FUNCTION_BLOCK Master_TEST (* Composite Function Block Type *)
  (* Standard: 61499-2 *)
  (* Version 0.2, 2003-12-05, JHC, Rockwell Automation, Renamed from NEWCOMPFB. *)
  (* Version 0.1, 2002-01-08, JHC, Rockwell Automation, Added DLY FB as example. *)
  (* Version 0.0, 2000-05-27, JHC, Rockwell Automation *)
  (* Compiler header: package fb.rt.pnp; *)
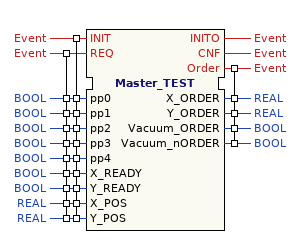
  EVENT_INPUT
    INIT WITH pp0, pp1, pp2, pp3, pp4, X_READY, Y_READY, X_POS, Y_POS; (* Initialization Request *)
    REQ WITH pp0, pp1, pp2, pp3, pp4, X_READY, Y_READY, X_POS, Y_POS; (* Normal Execution Request *)
  END_EVENT
  EVENT_OUTPUT
    INITO; (* Initialization Confirm *)
    CNF; (* Execution Confirmation *)
    Order WITH X_ORDER, Y_ORDER, Vacuum_ORDER, Vacuum_nORDER;
  END_EVENT
  VAR_INPUT
    pp0 : BOOL;
    pp1 : BOOL;
    pp2 : BOOL;
    pp3 : BOOL;
    pp4 : BOOL;
    X_READY : BOOL;
    Y_READY : BOOL;
    X_POS : REAL;
    Y_POS : REAL;
  END_VAR
  VAR_OUTPUT
    X_ORDER : REAL;
    Y_ORDER : REAL;
    Vacuum_ORDER : BOOL;
    Vacuum_nORDER : BOOL;
  END_VAR
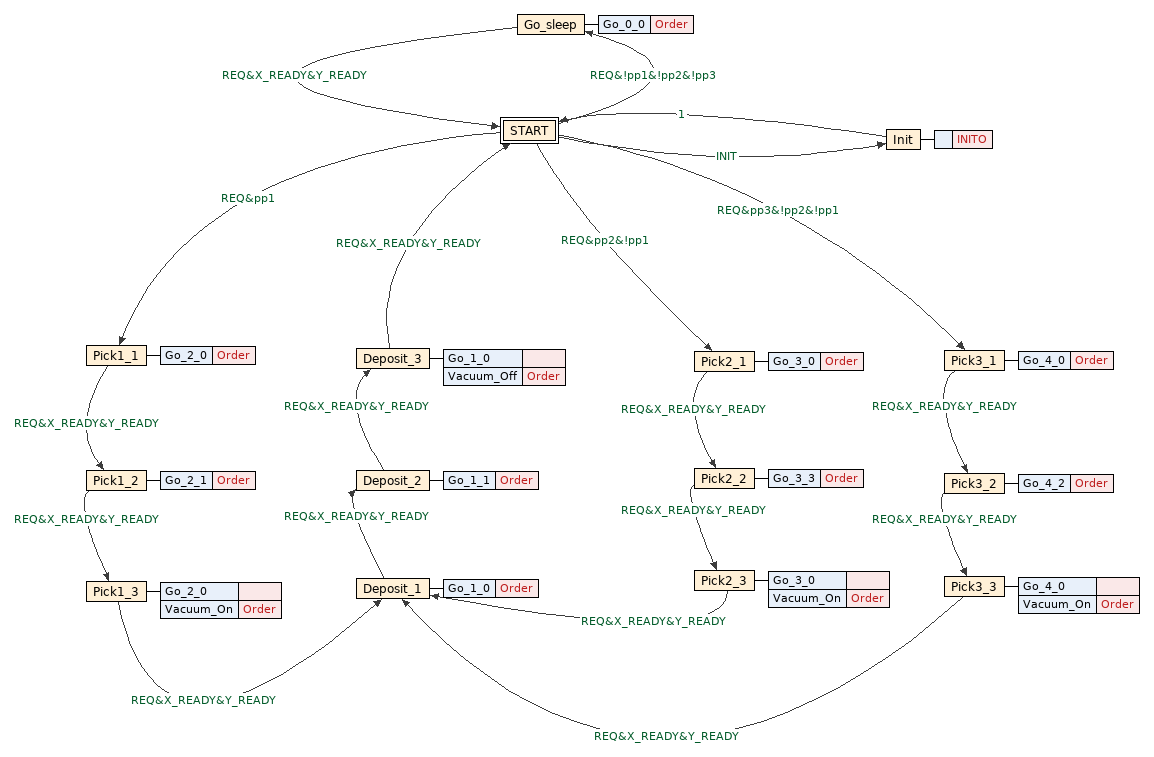
  EC_STATES
    START; (* Initial State *)
    Pick3_3 : Go_4_0, Vacuum_On -> Order;
    Pick3_1 : Go_4_0 -> Order;
    Pick3_2 : Go_4_2 -> Order;
    Pick2_3 : Go_3_0, Vacuum_On -> Order;
    Pick2_1 : Go_3_0 -> Order;
    Pick2_2 : Go_3_3 -> Order;
    Pick1_3 : Go_2_0, Vacuum_On -> Order;
    Pick1_1 : Go_2_0 -> Order;
    Pick1_2 : Go_2_1 -> Order;
    Deposit_1 : Go_1_0 -> Order;
    Deposit_2 : Go_1_1 -> Order;
    Deposit_3 : Go_1_0, Vacuum_Off -> Order;
    Go_sleep : Go_0_0 -> Order;
    Init : -> INITO;
  END_STATES
  EC_TRANSITIONS
    START TO Pick1_1 := REQ&pp1;
    Pick1_1 TO Pick1_2 := REQ&X_READY&Y_READY;
    Pick1_2 TO Pick1_3 := REQ&X_READY&Y_READY;
    Pick1_3 TO Deposit_1 := REQ&X_READY&Y_READY;
    Deposit_1 TO Deposit_2 := REQ&X_READY&Y_READY;
    Deposit_2 TO Deposit_3 := REQ&X_READY&Y_READY;
    Deposit_3 TO START := REQ&X_READY&Y_READY;
    START TO Pick2_1 := REQ&pp2&!pp1;
    START TO Pick3_1 := REQ&pp3&!pp2&!pp1;
    Pick2_1 TO Pick2_2 := REQ&X_READY&Y_READY;
    Pick2_2 TO Pick2_3 := REQ&X_READY&Y_READY;
    Pick3_1 TO Pick3_2 := REQ&X_READY&Y_READY;
    Pick3_2 TO Pick3_3 := REQ&X_READY&Y_READY;
    Pick3_3 TO Deposit_1 := REQ&X_READY&Y_READY;
    Pick2_3 TO Deposit_1 := REQ&X_READY&Y_READY;
    Go_sleep TO START := REQ&X_READY&Y_READY;
    START TO Go_sleep := REQ&!pp1&!pp2&!pp3;
    START TO Init := INIT;
    Init TO START := 1;
  END_TRANSITIONS
  ALGORITHM INIT IN Java: (* Initialization algorithm *)
System.out.println("init!!!");
  END_ALGORITHM
  ALGORITHM Vacuum_On IN Java: (* Normally executed algorithm *)
Vacuum_ORDER.value=true;
Vacuum_nORDER.value=false;
  END_ALGORITHM
  ALGORITHM Vacuum_Off IN Java: (* Normally executed algorithm *)
Vacuum_ORDER.value=false;
Vacuum_nORDER.value=true;
  END_ALGORITHM
  ALGORITHM Go_0_0 IN Java: (* Normally executed algorithm *)
X_ORDER.value=0;
Y_ORDER.value=0;
  END_ALGORITHM
  ALGORITHM Go_1_0 IN Java: (* Normally executed algorithm *)
X_ORDER.value=1;
Y_ORDER.value=0;
  END_ALGORITHM
  ALGORITHM Go_2_0 IN Java: (* Normally executed algorithm *)
X_ORDER.value=2;
Y_ORDER.value=0;
  END_ALGORITHM
  ALGORITHM Go_3_0 IN Java: (* Normally executed algorithm *)
X_ORDER.value=3;
Y_ORDER.value=0;
  END_ALGORITHM
  ALGORITHM Go_4_0 IN Java: (* Normally executed algorithm *)
X_ORDER.value=4;
Y_ORDER.value=0;
  END_ALGORITHM
  ALGORITHM Go_1_1 IN Java: (* Normally executed algorithm *)
X_ORDER.value=1;
Y_ORDER.value=1;
  END_ALGORITHM
  ALGORITHM Go_2_1 IN Java: (* Normally executed algorithm *)
X_ORDER.value=2;
Y_ORDER.value=1;
  END_ALGORITHM
  ALGORITHM Go_3_3 IN Java: (* Normally executed algorithm *)
X_ORDER.value=3;
Y_ORDER.value=3;
  END_ALGORITHM
  ALGORITHM Go_4_2 IN Java: (* Normally executed algorithm *)
X_ORDER.value=4;
Y_ORDER.value=2;
  END_ALGORITHM
END_FUNCTION_BLOCK
